PROGRAM MAIN
VAR
	bEnable : BOOL;
	bStart : BOOL;
END_VAR

bEnable := bStart;

END_PROGRAM

(* stored: Version 1.1.0.1, ProductVersion 3.1.4024.12
   POU MAIN: Id {b4d41fb1-61e7-45bd-8077-0e67631c1f8f}, SpecialFunc None *)
